// TwinCAT 3 PLC project PLCSTD
// ProgramVersion: 3.1.4023.0
// libraries:
//   Tc2_MC2, * (Beckhoff Automation GmbH)
//   Tc2_MC2_Drive, * (Beckhoff Automation GmbH)
//   Tc2_Standard, * (Beckhoff Automation GmbH)
//   Tc2_System, * (Beckhoff Automation GmbH)
//   Tc2_Utilities, * (Beckhoff Automation GmbH)
//   Tc3_Module, * (Beckhoff Automation GmbH)
// project tree:
//   DUTs/ ST_MC_CMD.TcDUT, ST_MC_Status.TcDUT
//   GVLs/ GVL_SA.TcGVL
//   / PlcTask.TcTTO
//   POUs/ MAIN.TcPOU, MotionControl.TcPOU
// real-time tasks:
//   TASK PlcTask: cycle T#10ms, priority 20, ADS port 350
// motion (NC):
//   TASK NC-Task 1 SAF: cycle T#2ms, priority 4, ADS port 501
//   TASK NC-Task 1 SVB: cycle T#10ms, priority 8, ADS port 511
//   AXIS Axis 1 (id 1)
//     OtherSettings: AllowMotionCmdToSlave=true
//     encoder EncType=19
//       EncPara: MaxCount=#xffffffff
//     drive DrvType=16
//       DrvPara: MaxCount=#xffffffff, DriveControlDWord=#x00020000
//         Analog: TorqueSetpointScale=10, ScaleFactorActTorque=0.1
//         TimeComp: TaskDelayCycles=1
//     controller CtrType=1
//       CtrPara: PriorControlFactor=1
//         Observer: BandWidth=20
//   AXIS Axis 2 (id 2)
//     OtherSettings: AllowMotionCmdToSlave=true
//     encoder EncType=7
//       EncPara: MaxCount=#x0000ffff, ReferenceSystem=1
//     drive DrvType=5
//       Analog: TorqueSetpointScale=10, ScaleFactorActTorque=0.1
//       TimeComp: TaskDelayCycles=1
//     controller CtrType=2
//       CtrPara: PriorControlFactor=1
//         Observer: BandWidth=20
//   AXIS Axis 3 Virtual (id 3)
//     OtherSettings: AllowMotionCmdToSlave=true
//     encoder EncType=1
//     drive DrvType=5
//       Analog: TorqueSetpointScale=10, ScaleFactorActTorque=0.1
//       TimeComp: TaskDelayCycles=1
//     controller CtrType=1
//       CtrPara: PriorControlFactor=1
//         Observer: BandWidth=20
// I/O:
//   DEVICE Device 1 (EtherCAT) (disabled), AmsNetId 192.168.0.100.2.1
//     Term 1 (EK1200) [EK1200-5000 EtherCAT Power supply (2A E-Bus)]
//       Term 2 (EL1008) [EL1008 8Ch. Dig. Input 24V, 3ms]
//       Term 3 (EL2008) [EL2008 8Ch. Dig. Output 24V, 0.5A]
//       Drive 4 (EL7201-0001) [EL7201-0001 1Ch. DS402 Servo motor output stage (50V, 4A)]
//       Term 5 (EL3042) [EL3042 2Ch. Ana. Input 0-20mA]
//       Term 6 (EL4012) [EL4012 2Ch. Ana. Output 0-20mA, 12bit]
//       Term 7 (EK1122) [EK1122 2 port EtherCAT junction]
// variable links:
//   NC-Task 1 SAF/Axes/Axis 1 <-> Device 1 (EtherCAT)/Term 1 (EK1200)/Drive 4 (EL7201-0001)
//     Drive/Inputs/In/nDcOutputTime <-> InfoData/DcOutputShift
//     Drive/Inputs/In/nState1 <-> DS402 Statusword/Statusword
//     Drive/Inputs/In/nState2 <-> DS402 Statusword/Statusword @bit 8
//     Drive/Inputs/In/nState4 @bit 1 <-> WcState/InputToggle
//     Drive/Inputs/In/nState4 <-> WcState/WcState
//     Drive/Outputs/Out/nCtrl1 <-> DS402 Controlword/Controlword
//     Drive/Outputs/Out/nCtrl2 <-> DS402 Controlword/Controlword @bit 8
//     Drive/Outputs/Out/nDataOut2 <-> DS402 Target velocity/Target velocity
//     Enc/Inputs/In/nDataIn1 <-> DS402 Position actual value/Position actual value
//     Enc/Inputs/In/nDcInputTime <-> InfoData/DcInputShift
//     Enc/Inputs/In/nState4 @bit 1 <-> WcState/InputToggle
//     Enc/Inputs/In/nState4 <-> WcState/WcState
//   NC-Task 1 SAF/Axes/Axis 2 <-> Device 1 (EtherCAT)/Term 1 (EK1200)/Term 5 (EL3042)
//     Enc/Inputs/In/nDataIn1[0] <-> AI Standard Channel 2/Value
//     Enc/Inputs/In/nState4 @bit 1 <-> WcState/InputToggle
//     Enc/Inputs/In/nState4 <-> WcState/WcState
//   NC-Task 1 SAF/Axes/Axis 2 <-> Device 1 (EtherCAT)/Term 1 (EK1200)/Term 6 (EL4012)
//     Drive/Inputs/In/nState4 <-> WcState/WcState
//     Drive/Outputs/Out/nDataOut1[0] <-> AO Outputs Channel 1/Analog output
//   PLCSTD/PLCSTD Instance <-> NC-Task 1 SAF/Axes/Axis 3 Virtual
//     PlcTask Inputs/GVL_SA.SingleAxis.NcToPlc <-> Outputs/ToPlc
//     PlcTask Outputs/GVL_SA.SingleAxis.PlcToNc <-> Inputs/FromPlc

CONFIGURATION PLCSTD
    RESOURCE PLC ON TwinCAT3
        TASK PlcTask(INTERVAL := T#10ms, PRIORITY := 20);
        PROGRAM MAIN WITH PlcTask : MAIN;
    END_RESOURCE
END_CONFIGURATION

// ---- DUTs/ST_MC_CMD.TcDUT
TYPE ST_MC_CMD :
STRUCT
	bExe			:BOOL;
	lrVelocity		:LREAL;
	lrAcceleration 	:LREAL;
	lrDeceleration 	:LREAL;
	lrJerk		 	:LREAL;
	lrDistance	 	:LREAL;
	lrPosition	 	:LREAL;
	EnuDirection	:MC_Direction;
	EnuBufferMode	:MC_BufferMode;
	EnuOptions		:ST_MoveOptions;
	
	
END_STRUCT
END_TYPE

// ---- DUTs/ST_MC_Status.TcDUT
TYPE ST_MC_Status :
STRUCT
	
	Status		: BOOL;
	Done	 	: BOOL;
	Busy	 	: BOOL;
	Error	 	: BOOL;
	Active	 	: BOOL;
	CmdAborted 	: BOOL;
	InVelocity	: BOOL;
	errorID	 	: UDINT;
	
END_STRUCT
END_TYPE

// ---- GVLs/GVL_SA.TcGVL
{attribute 'qualified_only'}
VAR_GLOBAL
    //Single Axis
	SingleAxis : AXIS_REF;
	
	//Motino Control Function VLock Instant Variable 'fbSA'
	fbSA_Reset	: MC_Reset;
	fbSA_Power	: MC_Power;
	fbSA_Home	: MC_Home;
	fbSA_Jog	: MC_Jog;
	fbSA_MovVel1 : MC_MoveVelocity;
	fbSA_MovVel2 : MC_MoveVelocity;
	fbSA_MovRel1 : MC_MoveRelative;
	fbSA_MovRel2 : MC_MoveRelative;
	fbSA_MovAbs1 : MC_MoveAbsolute;
	fbSA_MovAbs2 : MC_MoveAbsolute;
	
	//	input: Command
	bSA_ResetExe		: BOOL;
	
	bSA_PowerEnCmd		: BOOL;
	bSA_PowerEnPositive	: BOOL;
	bSA_PowerEnNegative : BOOL;
	
	bSA_HomeExe			: BOOL;
	bSA_HomeCamInput	: BOOL;
	
	bSA_JogFwd			: BOOL;
	bSA_JogRev			: BOOL;
	
	stSA_VelCmd1			: ST_MC_CMD;
	stSA_VelCmd2			: ST_MC_CMD;
	stSA_RelCmd1			: ST_MC_CMD;
	stSA_RelCmd2			: ST_MC_CMD;
	stSA_AbsCmd1 			: ST_MC_CMD;
	stSA_AbsCmd2			: ST_MC_CMD;
	
	//Variable PArameters
	lrSA_PowerOverride	:LREAL;
	lrSA_HomePosition	:LREAL;
	lrSA_SetPosition	:LREAL;
	lrSA_JogVelocity	:LREAL;
	
	
	//Status
	stSA_Reset			: ST_MC_Status;
	stSA_Power			: ST_MC_Status;
	stSA_Home			: ST_MC_Status;
	stSA_SetPosition	: ST_MC_Status;
	stSA_Jog			: ST_MC_Status;
	
	stSA_VelSts1		: ST_MC_Status;
	stSA_VelSts2		: ST_MC_Status;
	stSA_RelSts1		: ST_MC_Status;
	stSA_RelSts2		: ST_MC_Status;
	stSA_AbsSts1		: ST_MC_Status;
	stSA_AbsSts2		: ST_MC_Status;
	
END_VAR

// ---- POUs/MAIN.TcPOU
PROGRAM MAIN
VAR
END_VAR

MotionControl();

END_PROGRAM

// ---- POUs/MotionControl.TcPOU
PROGRAM MotionControl
VAR
END_VAR

SingleAxis_LD();

METHOD SingleAxis_LD : BOOL
VAR_INPUT
END_VAR
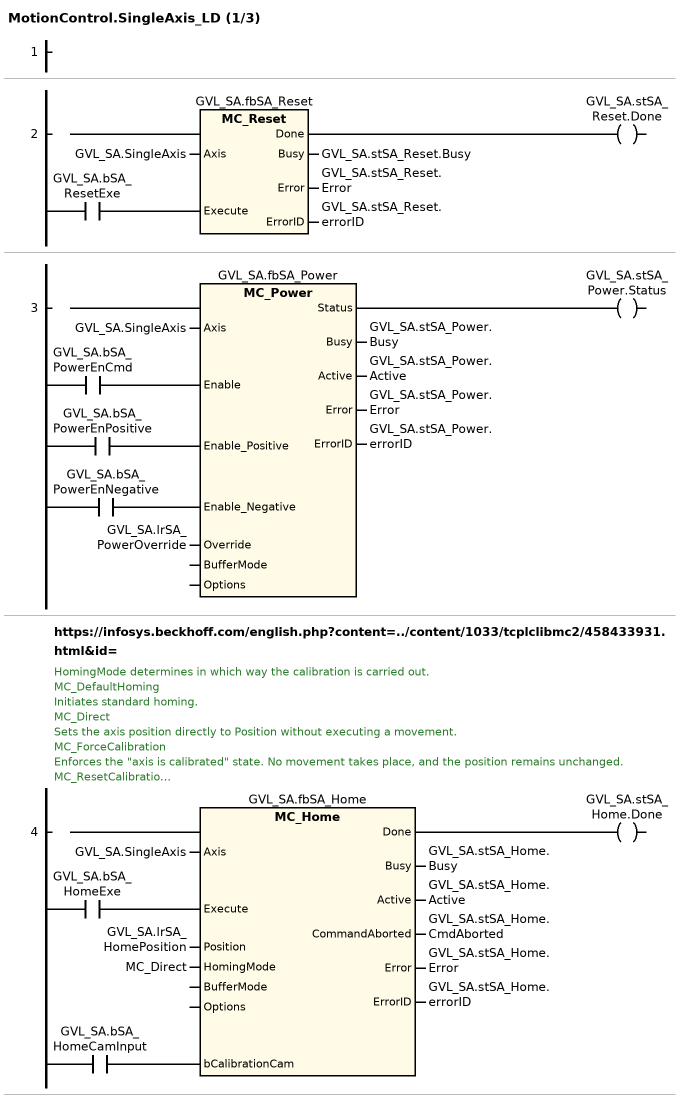
// NETWORK 1

// NETWORK 2
GVL_SA.fbSA_Reset(
    Axis := GVL_SA.SingleAxis,
    Execute := GVL_SA.bSA_ResetExe,
    Busy => GVL_SA.stSA_Reset.Busy,
    Error => GVL_SA.stSA_Reset.Error,
    ErrorID => GVL_SA.stSA_Reset.errorID); // MC_Reset
GVL_SA.stSA_Reset.Done := GVL_SA.fbSA_Reset.Done;

// NETWORK 3
GVL_SA.fbSA_Power(
    Axis := GVL_SA.SingleAxis,
    Enable := GVL_SA.bSA_PowerEnCmd,
    Enable_Positive := GVL_SA.bSA_PowerEnPositive,
    Enable_Negative := GVL_SA.bSA_PowerEnNegative,
    Override := GVL_SA.lrSA_PowerOverride,
    Busy => GVL_SA.stSA_Power.Busy,
    Active => GVL_SA.stSA_Power.Active,
    Error => GVL_SA.stSA_Power.Error,
    ErrorID => GVL_SA.stSA_Power.errorID); // MC_Power
GVL_SA.stSA_Power.Status := GVL_SA.fbSA_Power.Status;

// NETWORK 4: https://infosys.beckhoff.com/english.php?content=../content/1033/tcplclibmc2/458433931.html&id=
// HomingMode determines in which way the calibration is carried out.
//
// MC_DefaultHoming
// Initiates standard homing.
// MC_Direct
// Sets the axis position directly to Position without executing a movement.
// MC_ForceCalibration
// Enforces the "axis is calibrated" state. No movement takes place, and the position remains unchanged.
// MC_ResetCalibration
// Resets the calibration state of the axis. No movement takes place, and the position remains unchanged.
GVL_SA.fbSA_Home(
    Axis := GVL_SA.SingleAxis,
    Execute := GVL_SA.bSA_HomeExe,
    Position := GVL_SA.lrSA_HomePosition,
    HomingMode := MC_Direct,
    bCalibrationCam := GVL_SA.bSA_HomeCamInput,
    Busy => GVL_SA.stSA_Home.Busy,
    Active => GVL_SA.stSA_Home.Active,
    CommandAborted => GVL_SA.stSA_Home.CmdAborted,
    Error => GVL_SA.stSA_Home.Error,
    ErrorID => GVL_SA.stSA_Home.errorID); // MC_Home
GVL_SA.stSA_Home.Done := GVL_SA.fbSA_Home.Done;

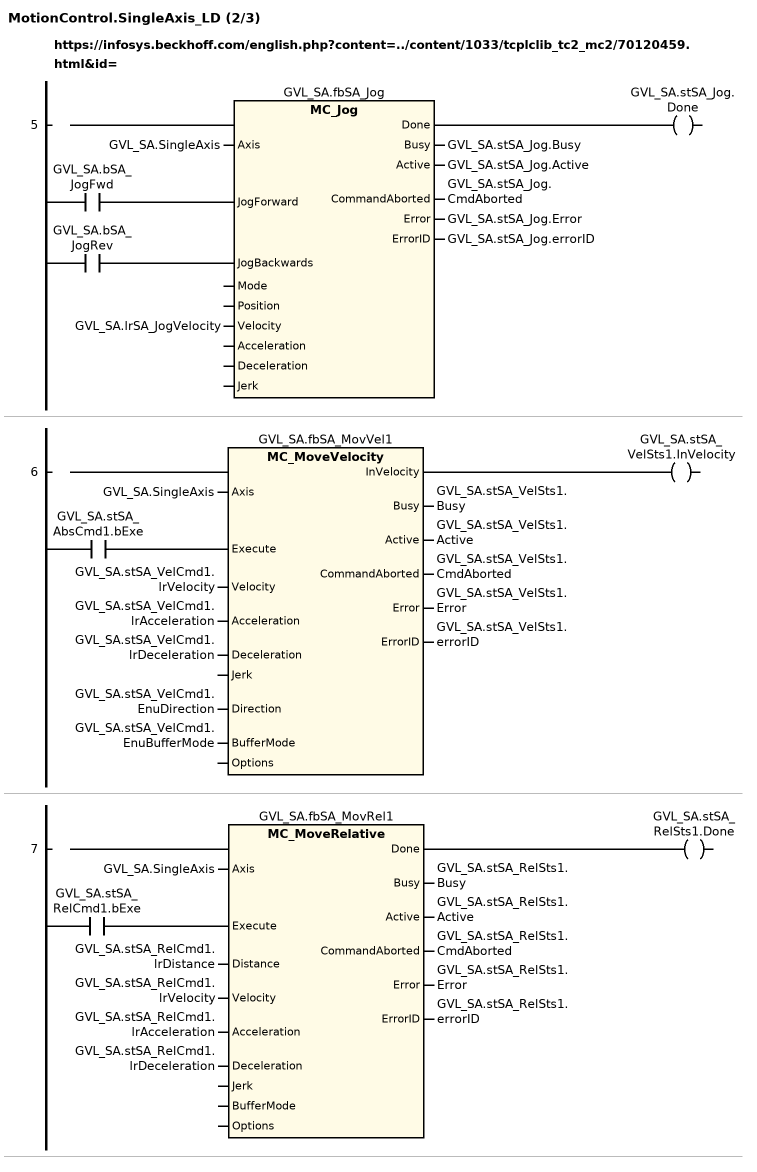
// NETWORK 5: https://infosys.beckhoff.com/english.php?content=../content/1033/tcplclib_tc2_mc2/70120459.html&id=
GVL_SA.fbSA_Jog(
    Axis := GVL_SA.SingleAxis,
    JogForward := GVL_SA.bSA_JogFwd,
    JogBackwards := GVL_SA.bSA_JogRev,
    Velocity := GVL_SA.lrSA_JogVelocity,
    Busy => GVL_SA.stSA_Jog.Busy,
    Active => GVL_SA.stSA_Jog.Active,
    CommandAborted => GVL_SA.stSA_Jog.CmdAborted,
    Error => GVL_SA.stSA_Jog.Error,
    ErrorID => GVL_SA.stSA_Jog.errorID); // MC_Jog
GVL_SA.stSA_Jog.Done := GVL_SA.fbSA_Jog.Done;

// NETWORK 6
GVL_SA.fbSA_MovVel1(
    Axis := GVL_SA.SingleAxis,
    Execute := GVL_SA.stSA_AbsCmd1.bExe,
    Velocity := GVL_SA.stSA_VelCmd1.lrVelocity,
    Acceleration := GVL_SA.stSA_VelCmd1.lrAcceleration,
    Deceleration := GVL_SA.stSA_VelCmd1.lrDeceleration,
    Direction := GVL_SA.stSA_VelCmd1.EnuDirection,
    BufferMode := GVL_SA.stSA_VelCmd1.EnuBufferMode,
    Busy => GVL_SA.stSA_VelSts1.Busy,
    Active => GVL_SA.stSA_VelSts1.Active,
    CommandAborted => GVL_SA.stSA_VelSts1.CmdAborted,
    Error => GVL_SA.stSA_VelSts1.Error,
    ErrorID => GVL_SA.stSA_VelSts1.errorID); // MC_MoveVelocity
GVL_SA.stSA_VelSts1.InVelocity := GVL_SA.fbSA_MovVel1.InVelocity;

// NETWORK 7
GVL_SA.fbSA_MovRel1(
    Axis := GVL_SA.SingleAxis,
    Execute := GVL_SA.stSA_RelCmd1.bExe,
    Distance := GVL_SA.stSA_RelCmd1.lrDistance,
    Velocity := GVL_SA.stSA_RelCmd1.lrVelocity,
    Acceleration := GVL_SA.stSA_RelCmd1.lrAcceleration,
    Deceleration := GVL_SA.stSA_RelCmd1.lrDeceleration,
    Busy => GVL_SA.stSA_RelSts1.Busy,
    Active => GVL_SA.stSA_RelSts1.Active,
    CommandAborted => GVL_SA.stSA_RelSts1.CmdAborted,
    Error => GVL_SA.stSA_RelSts1.Error,
    ErrorID => GVL_SA.stSA_RelSts1.errorID); // MC_MoveRelative
GVL_SA.stSA_RelSts1.Done := GVL_SA.fbSA_MovRel1.Done;

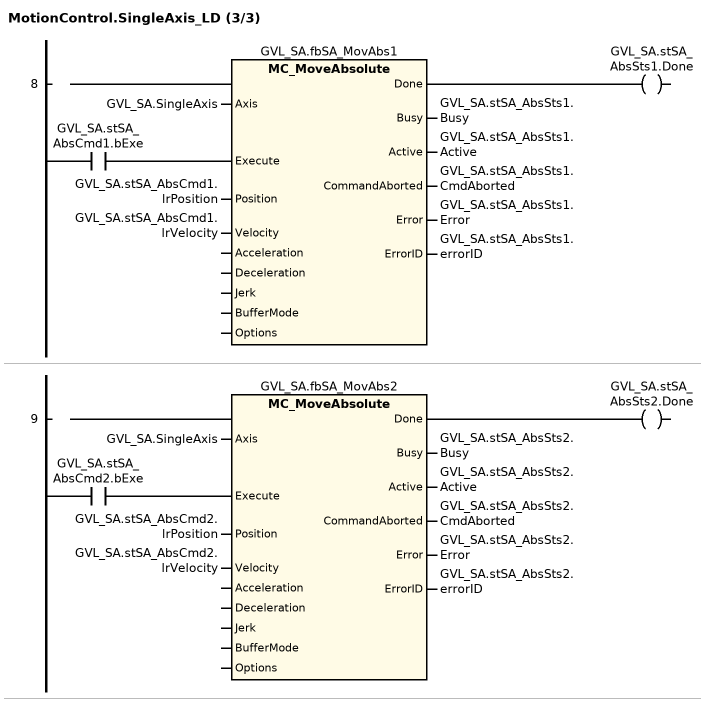
// NETWORK 8
GVL_SA.fbSA_MovAbs1(
    Axis := GVL_SA.SingleAxis,
    Execute := GVL_SA.stSA_AbsCmd1.bExe,
    Position := GVL_SA.stSA_AbsCmd1.lrPosition,
    Velocity := GVL_SA.stSA_AbsCmd1.lrVelocity,
    Busy => GVL_SA.stSA_AbsSts1.Busy,
    Active => GVL_SA.stSA_AbsSts1.Active,
    CommandAborted => GVL_SA.stSA_AbsSts1.CmdAborted,
    Error => GVL_SA.stSA_AbsSts1.Error,
    ErrorID => GVL_SA.stSA_AbsSts1.errorID); // MC_MoveAbsolute
GVL_SA.stSA_AbsSts1.Done := GVL_SA.fbSA_MovAbs1.Done;

// NETWORK 9
GVL_SA.fbSA_MovAbs2(
    Axis := GVL_SA.SingleAxis,
    Execute := GVL_SA.stSA_AbsCmd2.bExe,
    Position := GVL_SA.stSA_AbsCmd2.lrPosition,
    Velocity := GVL_SA.stSA_AbsCmd2.lrVelocity,
    Busy => GVL_SA.stSA_AbsSts2.Busy,
    Active => GVL_SA.stSA_AbsSts2.Active,
    CommandAborted => GVL_SA.stSA_AbsSts2.CmdAborted,
    Error => GVL_SA.stSA_AbsSts2.Error,
    ErrorID => GVL_SA.stSA_AbsSts2.errorID); // MC_MoveAbsolute
GVL_SA.stSA_AbsSts2.Done := GVL_SA.fbSA_MovAbs2.Done;
END_METHOD

END_PROGRAM
